FUNCTION FC_SQL_InsertCommands_TempSensor : STRING(255)
VAR_INPUT
    iSensorValue: STRING;
    iSampleNr: INT;
	iSensorID: INT;
	iMeasurementNr: INT;
END_VAR

FC_SQL_InsertCommands_TempSensor := 'INSERT INTO [db_accessadmin].[TempSensor] (SensorValue, SampleNr, Time, SensorID, MeasurementNr) VALUES (';
FC_SQL_InsertCommands_TempSensor := CONCAT(FC_SQL_InsertCommands_TempSensor, iSensorValue);
FC_SQL_InsertCommands_TempSensor := CONCAT(FC_SQL_InsertCommands_TempSensor, ', ');
FC_SQL_InsertCommands_TempSensor := CONCAT(FC_SQL_InsertCommands_TempSensor, INT_TO_STRING(iSampleNr));
FC_SQL_InsertCommands_TempSensor := CONCAT(FC_SQL_InsertCommands_TempSensor, ', GETDATE(), ');
FC_SQL_InsertCommands_TempSensor := CONCAT(FC_SQL_InsertCommands_TempSensor, INT_TO_STRING(iSensorID));
FC_SQL_InsertCommands_TempSensor := CONCAT(FC_SQL_InsertCommands_TempSensor, ', ');
FC_SQL_InsertCommands_TempSensor := CONCAT(FC_SQL_InsertCommands_TempSensor, INT_TO_STRING(iMeasurementNr));
FC_SQL_InsertCommands_TempSensor := CONCAT(FC_SQL_InsertCommands_TempSensor, ');');

END_FUNCTION

(* stored: Version 1.1.0.1
   POU FC_SQL_InsertCommands_TempSensor: Id {679b0b15-8183-47b4-b50a-239f76f313e1}, SpecialFunc None *)
